FUNCTION_BLOCK fbManipulatorAutomat EXTENDS TcoCore.TcoState
VAR
	_horizontalPiston : fbPiston(THIS^);
	_verticalPiston : fbPiston(THIS^);
	_gripperPiston : fbPiston(THIS^);
END_VAR

_horizontalPiston();
_verticalPiston();
_gripperPiston();

IF(THIS^.State = 0) THEN	
	IF(_verticalPiston.MoveHome().Done 
		AND_THEN _horizontalPiston.MoveHome().Done 
		AND_THEN _gripperPiston.MoveHome().Done) THEN
		THIS^.ChangeState(10);
	END_IF
END_IF

IF(THIS^.State = 10) THEN
	IF(_verticalPiston.MoveWork().Done) THEN
		THIS^.ChangeState(20);
	END_IF
END_IF

IF(THIS^.State = 20) THEN
	IF(_gripperPiston.MoveWork().Done) THEN
		THIS^.ChangeState(30);
	END_IF
END_IF

IF(THIS^.State = 30) THEN
	IF(_verticalPiston.MoveHome().Done) THEN
		THIS^.ChangeState(40);
	END_IF
END_IF

IF(THIS^.State = 40) THEN
	IF(_horizontalPiston.MoveWork().Done) THEN
		THIS^.ChangeState(50);
	END_IF
END_IF

IF(THIS^.State = 50) THEN
	IF(_verticalPiston.MoveWork().Done) THEN
		THIS^.ChangeState(60);
	END_IF
END_IF

IF(THIS^.State = 60) THEN
	IF(_gripperPiston.MoveHome().Done) THEN
		THIS^.ChangeState(0);
	END_IF
END_IF

END_FUNCTION_BLOCK

(* stored: Version 1.1.0.1, ProductVersion 3.1.4024.6
   POU fbManipulatorAutomat: Id {1e6d1f44-12f8-4565-9151-b2b01976380d}, SpecialFunc None *)
